{attribute addProperty BoxType "EP8309-0022-0021"}
{attribute addProperty Id "StatusAT %I*Status_D7D8B361162"}
{attribute addProperty CRC "502109842"}
{attribute addProperty SizeInBites "16"}
{attribute addProperty SizeInBytes "2"}
TYPE PWM_Status_1DED9692 :
STRUCT
	{attribute addProperty Name "Status"}
	Status AT %I* : Status_D7D8B361;
END_STRUCT
END_TYPE

(* stored: Version 1.2.0.0, ProductVersion 3.1.4024.9
   DUT PWM_Status_1DED9692: Id {aca864b2-cb3b-41e0-bac8-e403ed5bcd38} *)
